// TIA Portal V19 export
DATA_BLOCK "FinalCutLub_PERS"   // DB218
{ DB_Accessible_From_OPC_UA := 'FALSE' }
// stored: DBAccessibleFromOPCUA false, MemoryReserve 100
   VAR RETAIN
      PersistentValues : Struct
         Data : Struct
            SavedCutBenchCode : DInt := 0;
            PumpJobCounter : UDInt := 0;
            JobsCounter : UDInt := 0;
         END_STRUCT;
         Par : Struct
            SystemOffOn : Bool := TRUE;
            JobsToStart : UDInt := 15;
            OilPumpCycles : UDInt := 10;
         END_STRUCT;
      END_STRUCT;
   END_VAR
BEGIN
END_DATA_BLOCK
